Yaskawa INFORM job: MAX_BACK_7.JBI

/JOB
//NAME MAX_BACK_7
///FOLDERNAME INTERNE_BERECHNUNGEN
//POS
///NPOS 0,0,0,0,0,0
//ALIAS
///LVARS 0,0,7,0,0,0,0,0
LD000 VAL_MAX
LD001 VAL_2
LD002 VAL_3
LD003 VAL_4
LD004 VAL_5
LD005 VAL_6
LD006 VAL_7
//ARGINFO
///ARGTYPE D,D,D,D,D,D,D,
///COMMENT
VALUE_IN_1
VALUE_IN_2
VALUE_IN_3
VALUE_IN_4
VALUE_IN_5
VALUE_IN_6
VALUE_IN_7

//INST
///DATE 2021/10/11 09:26
///COMM Gives back max value out of 7
///ATTR SC,RW
///LVARS 0,0,7,0,0,0,0,0
NOP
GETARG VAL_MAX IARG#(1)
GETARG VAL_2 IARG#(2)
GETARG VAL_3 IARG#(3)
GETARG VAL_4 IARG#(4)
GETARG VAL_5 IARG#(5)
GETARG VAL_6 IARG#(6)
GETARG VAL_7 IARG#(7)
'################################
'MINIMALHOEHE BESTIMMEN
IFTHENEXP VAL_2>VAL_MAX
	 SET VAL_MAX VAL_2
ENDIF
IFTHENEXP VAL_3>VAL_MAX
	 SET VAL_MAX VAL_3
ENDIF
IFTHENEXP VAL_4>VAL_MAX
	 SET VAL_MAX VAL_4
ENDIF
IFTHENEXP VAL_5>VAL_MAX
	 SET VAL_MAX VAL_5
ENDIF
IFTHENEXP VAL_6>VAL_MAX
	 SET VAL_MAX VAL_6
ENDIF
IFTHENEXP VAL_7>VAL_MAX
	 SET VAL_MAX VAL_7
ENDIF
RET VAL_MAX
END
